// TIA Portal V20 export
// export: Created 2026-10-06T14:13:36.952242Z, ExportSetting WithDefaults, DisplayName Totally Integrated Automation Portal, DisplayVersion V20, DisplayName TIA Portal Openness, DisplayVersion V20, DisplayName TIA Portal Version Control Interface, DisplayVersion V20, DisplayName SINAMICS Startdrive Advanced, DisplayVersion V20, DisplayName SINAMICS Startdrive G130, G150, S120, S150, SINAMICS MV, G220, S200, S210, DisplayVersion V20, DisplayName SINAMICS Startdrive G110M, G120, G120C, G120D, G120P, G115D, DisplayVersion V20, DisplayName STEP 7 Professional, DisplayVersion V20, DisplayName STEP 7 Safety, DisplayVersion V20, DisplayName WinCC Basic/Comfort/Advanced, DisplayVersion V20, DisplayName WinCC Unified, DisplayVersion V20
FUNCTION_BLOCK "MotorSequenceLAD"   // FB1, LAD
{ S7_Optimized_Access := 'TRUE' }
VERSION : 0.1
// stored: AutoNumber true, IsIECCheckEnabled false, IsRetainMemResEnabled false, MemoryReserve 100, SetENOAutomatically false, UDAEnableTagReadback false
   VAR
      Start2 { S7_SetPoint := 'True'} : TON_TIME;
      Start3 { S7_SetPoint := 'True'} : TON_TIME;
      Stop2 { S7_SetPoint := 'True'} : TON_TIME;
      Stop1 { S7_SetPoint := 'True'} : TON_TIME;
   END_VAR
BEGIN

REGION Network 1: 启动上升沿，仅接受新的按钮动作
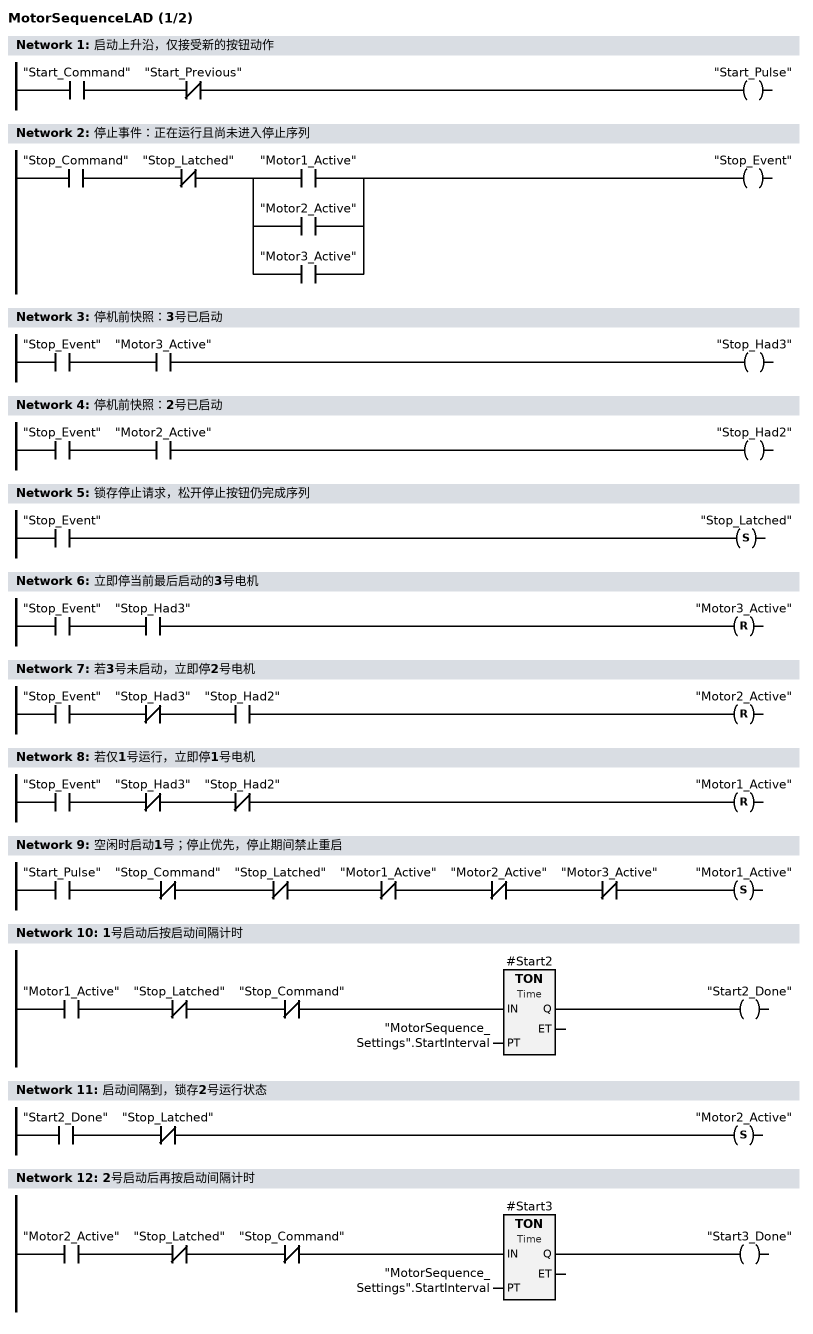
   RUNG wire#powerrail
      Contact( "Start_Command" )
      I_Contact( "Start_Previous" )
      Coil( "Start_Pulse" )
   END_RUNG
   // the same network as SCL:
   "Start_Pulse" := "Start_Command" AND NOT "Start_Previous";
END_REGION

REGION Network 2: 停止事件：正在运行且尚未进入停止序列
   RUNG wire#powerrail
      Contact( "Stop_Command" )
      I_Contact( "Stop_Latched" )
      wire#w1
      Contact( "Motor1_Active" )
      wire#w2
      Coil( "Stop_Event" )
   END_RUNG
   RUNG wire#w1
      Contact( "Motor2_Active" )
   END_RUNG wire#w2
   RUNG wire#w1
      Contact( "Motor3_Active" )
   END_RUNG wire#w2
   // the same network as SCL:
   "Stop_Event" := "Stop_Command" AND NOT "Stop_Latched" AND ("Motor1_Active" OR "Motor2_Active" OR "Motor3_Active");
END_REGION

REGION Network 3: 停机前快照：3号已启动
   RUNG wire#powerrail
      Contact( "Stop_Event" )
      Contact( "Motor3_Active" )
      Coil( "Stop_Had3" )
   END_RUNG
   // the same network as SCL:
   "Stop_Had3" := "Stop_Event" AND "Motor3_Active";
END_REGION

REGION Network 4: 停机前快照：2号已启动
   RUNG wire#powerrail
      Contact( "Stop_Event" )
      Contact( "Motor2_Active" )
      Coil( "Stop_Had2" )
   END_RUNG
   // the same network as SCL:
   "Stop_Had2" := "Stop_Event" AND "Motor2_Active";
END_REGION

REGION Network 5: 锁存停止请求，松开停止按钮仍完成序列
   RUNG wire#powerrail
      Contact( "Stop_Event" )
      S_Coil( "Stop_Latched" )
   END_RUNG
   // the same network as SCL:
   IF "Stop_Event" THEN "Stop_Latched" := TRUE; END_IF;
END_REGION

REGION Network 6: 立即停当前最后启动的3号电机
   RUNG wire#powerrail
      Contact( "Stop_Event" )
      Contact( "Stop_Had3" )
      R_Coil( "Motor3_Active" )
   END_RUNG
   // the same network as SCL:
   IF "Stop_Event" AND "Stop_Had3" THEN "Motor3_Active" := FALSE; END_IF;
END_REGION

REGION Network 7: 若3号未启动，立即停2号电机
   RUNG wire#powerrail
      Contact( "Stop_Event" )
      I_Contact( "Stop_Had3" )
      Contact( "Stop_Had2" )
      R_Coil( "Motor2_Active" )
   END_RUNG
   // the same network as SCL:
   IF "Stop_Event" AND NOT "Stop_Had3" AND "Stop_Had2" THEN "Motor2_Active" := FALSE; END_IF;
END_REGION

REGION Network 8: 若仅1号运行，立即停1号电机
   RUNG wire#powerrail
      Contact( "Stop_Event" )
      I_Contact( "Stop_Had3" )
      I_Contact( "Stop_Had2" )
      R_Coil( "Motor1_Active" )
   END_RUNG
   // the same network as SCL:
   IF "Stop_Event" AND NOT "Stop_Had3" AND NOT "Stop_Had2" THEN "Motor1_Active" := FALSE; END_IF;
END_REGION

REGION Network 9: 空闲时启动1号；停止优先，停止期间禁止重启
   RUNG wire#powerrail
      Contact( "Start_Pulse" )
      I_Contact( "Stop_Command" )
      I_Contact( "Stop_Latched" )
      I_Contact( "Motor1_Active" )
      I_Contact( "Motor2_Active" )
      I_Contact( "Motor3_Active" )
      S_Coil( "Motor1_Active" )
   END_RUNG
   // the same network as SCL:
   IF "Start_Pulse" AND NOT "Stop_Command" AND NOT "Stop_Latched" AND NOT "Motor1_Active" AND NOT "Motor2_Active" AND NOT "Motor3_Active" THEN
       "Motor1_Active" := TRUE;
   END_IF;
END_REGION

REGION Network 10: 1号启动后按启动间隔计时
   RUNG wire#powerrail
      Contact( "Motor1_Active" )
      I_Contact( "Stop_Latched" )
      I_Contact( "Stop_Command" )
      { S7_Templates := "time_type := Time" } #Start2.TON(pt := "MotorSequence_Settings".StartInterval, et =>)
      Coil( "Start2_Done" )
   END_RUNG
   // the same network as SCL:
   #Start2(IN := "Motor1_Active" AND NOT "Stop_Latched" AND NOT "Stop_Command",   // TON
           PT := "MotorSequence_Settings".StartInterval);
   "Start2_Done" := #Start2.Q;
END_REGION

REGION Network 11: 启动间隔到，锁存2号运行状态
   RUNG wire#powerrail
      Contact( "Start2_Done" )
      I_Contact( "Stop_Latched" )
      S_Coil( "Motor2_Active" )
   END_RUNG
   // the same network as SCL:
   IF "Start2_Done" AND NOT "Stop_Latched" THEN "Motor2_Active" := TRUE; END_IF;
END_REGION

REGION Network 12: 2号启动后再按启动间隔计时
   RUNG wire#powerrail
      Contact( "Motor2_Active" )
      I_Contact( "Stop_Latched" )
      I_Contact( "Stop_Command" )
      { S7_Templates := "time_type := Time" } #Start3.TON(pt := "MotorSequence_Settings".StartInterval, et =>)
      Coil( "Start3_Done" )
   END_RUNG
   // the same network as SCL:
   #Start3(IN := "Motor2_Active" AND NOT "Stop_Latched" AND NOT "Stop_Command",   // TON
           PT := "MotorSequence_Settings".StartInterval);
   "Start3_Done" := #Start3.Q;
END_REGION

REGION Network 13: 启动间隔到，锁存3号运行状态
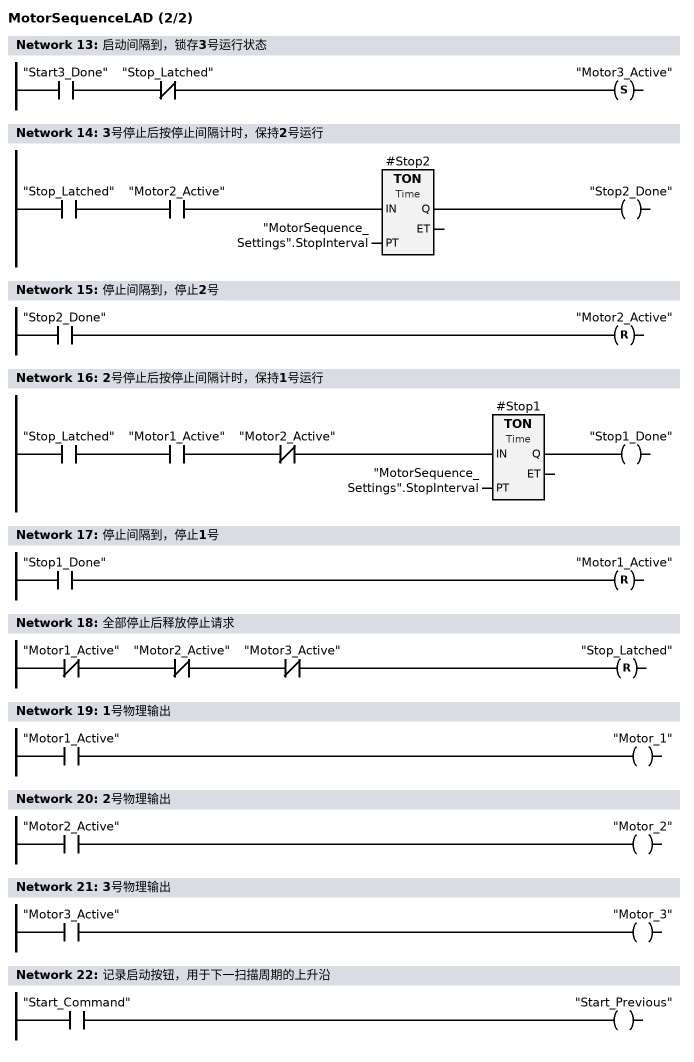
   RUNG wire#powerrail
      Contact( "Start3_Done" )
      I_Contact( "Stop_Latched" )
      S_Coil( "Motor3_Active" )
   END_RUNG
   // the same network as SCL:
   IF "Start3_Done" AND NOT "Stop_Latched" THEN "Motor3_Active" := TRUE; END_IF;
END_REGION

REGION Network 14: 3号停止后按停止间隔计时，保持2号运行
   RUNG wire#powerrail
      Contact( "Stop_Latched" )
      Contact( "Motor2_Active" )
      { S7_Templates := "time_type := Time" } #Stop2.TON(pt := "MotorSequence_Settings".StopInterval, et =>)
      Coil( "Stop2_Done" )
   END_RUNG
   // the same network as SCL:
   #Stop2(IN := "Stop_Latched" AND "Motor2_Active", PT := "MotorSequence_Settings".StopInterval);   // TON
   "Stop2_Done" := #Stop2.Q;
END_REGION

REGION Network 15: 停止间隔到，停止2号
   RUNG wire#powerrail
      Contact( "Stop2_Done" )
      R_Coil( "Motor2_Active" )
   END_RUNG
   // the same network as SCL:
   IF "Stop2_Done" THEN "Motor2_Active" := FALSE; END_IF;
END_REGION

REGION Network 16: 2号停止后按停止间隔计时，保持1号运行
   RUNG wire#powerrail
      Contact( "Stop_Latched" )
      Contact( "Motor1_Active" )
      I_Contact( "Motor2_Active" )
      { S7_Templates := "time_type := Time" } #Stop1.TON(pt := "MotorSequence_Settings".StopInterval, et =>)
      Coil( "Stop1_Done" )
   END_RUNG
   // the same network as SCL:
   #Stop1(IN := "Stop_Latched" AND "Motor1_Active" AND NOT "Motor2_Active",   // TON
          PT := "MotorSequence_Settings".StopInterval);
   "Stop1_Done" := #Stop1.Q;
END_REGION

REGION Network 17: 停止间隔到，停止1号
   RUNG wire#powerrail
      Contact( "Stop1_Done" )
      R_Coil( "Motor1_Active" )
   END_RUNG
   // the same network as SCL:
   IF "Stop1_Done" THEN "Motor1_Active" := FALSE; END_IF;
END_REGION

REGION Network 18: 全部停止后释放停止请求
   RUNG wire#powerrail
      I_Contact( "Motor1_Active" )
      I_Contact( "Motor2_Active" )
      I_Contact( "Motor3_Active" )
      R_Coil( "Stop_Latched" )
   END_RUNG
   // the same network as SCL:
   IF NOT "Motor1_Active" AND NOT "Motor2_Active" AND NOT "Motor3_Active" THEN
       "Stop_Latched" := FALSE;
   END_IF;
END_REGION

REGION Network 19: 1号物理输出
   RUNG wire#powerrail
      Contact( "Motor1_Active" )
      Coil( "Motor_1" )
   END_RUNG
   // the same network as SCL:
   "Motor_1" := "Motor1_Active";
END_REGION

REGION Network 20: 2号物理输出
   RUNG wire#powerrail
      Contact( "Motor2_Active" )
      Coil( "Motor_2" )
   END_RUNG
   // the same network as SCL:
   "Motor_2" := "Motor2_Active";
END_REGION

REGION Network 21: 3号物理输出
   RUNG wire#powerrail
      Contact( "Motor3_Active" )
      Coil( "Motor_3" )
   END_RUNG
   // the same network as SCL:
   "Motor_3" := "Motor3_Active";
END_REGION

REGION Network 22: 记录启动按钮，用于下一扫描周期的上升沿
   RUNG wire#powerrail
      Contact( "Start_Command" )
      Coil( "Start_Previous" )
   END_RUNG
   // the same network as SCL:
   "Start_Previous" := "Start_Command";
END_REGION
END_FUNCTION_BLOCK
